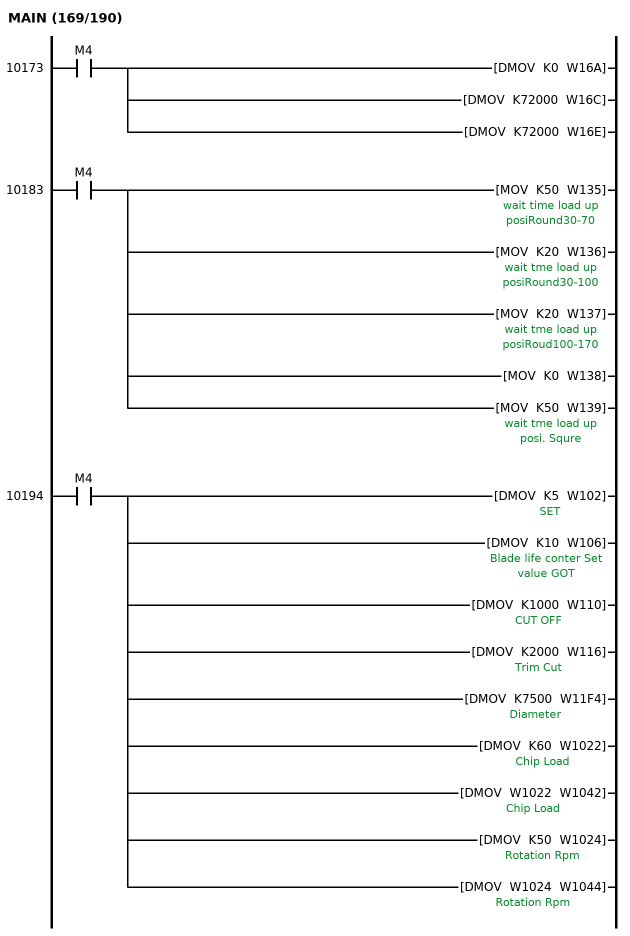
[picture p168: ladder of MAIN, rungs at steps 10173 to 10194]
10173 LD      M4
      DMOV    K0 W16A
      DMOV    K72000 W16C
      DMOV    K72000 W16E
10183 LD      M4
      MOV     K50 W135
      MOV     K20 W136
      MOV     K20 W137
      MOV     K0 W138
      MOV     K50 W139
10194 LD      M4
      DMOV    K5 W102
      DMOV    K10 W106
      DMOV    K1000 W110
      DMOV    K2000 W116
      DMOV    K7500 W11F4
      DMOV    K60 W1022
      DMOV    W1022 W1042
      DMOV    K50 W1024
      DMOV    W1024 W1044
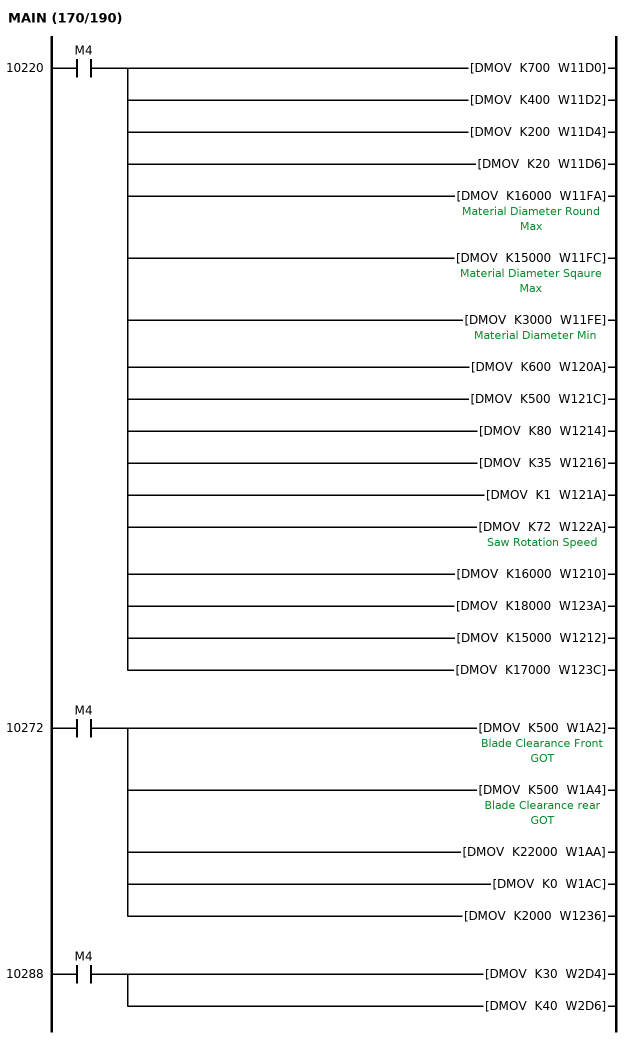
10220 LD      M4
      DMOV    K700 W11D0
      DMOV    K400 W11D2
      DMOV    K200 W11D4
      DMOV    K20 W11D6
      DMOV    K16000 W11FA
      DMOV    K15000 W11FC
      DMOV    K3000 W11FE
      DMOV    K600 W120A
      DMOV    K500 W121C
      DMOV    K80 W1214
      DMOV    K35 W1216
      DMOV    K1 W121A
      DMOV    K72 W122A
      DMOV    K16000 W1210
      DMOV    K18000 W123A
      DMOV    K15000 W1212
      DMOV    K17000 W123C
10272 LD      M4
      DMOV    K500 W1A2
      DMOV    K500 W1A4
      DMOV    K22000 W1AA
      DMOV    K0 W1AC
      DMOV    K2000 W1236
10288 LD      M4
      DMOV    K30 W2D4
      DMOV    K40 W2D6
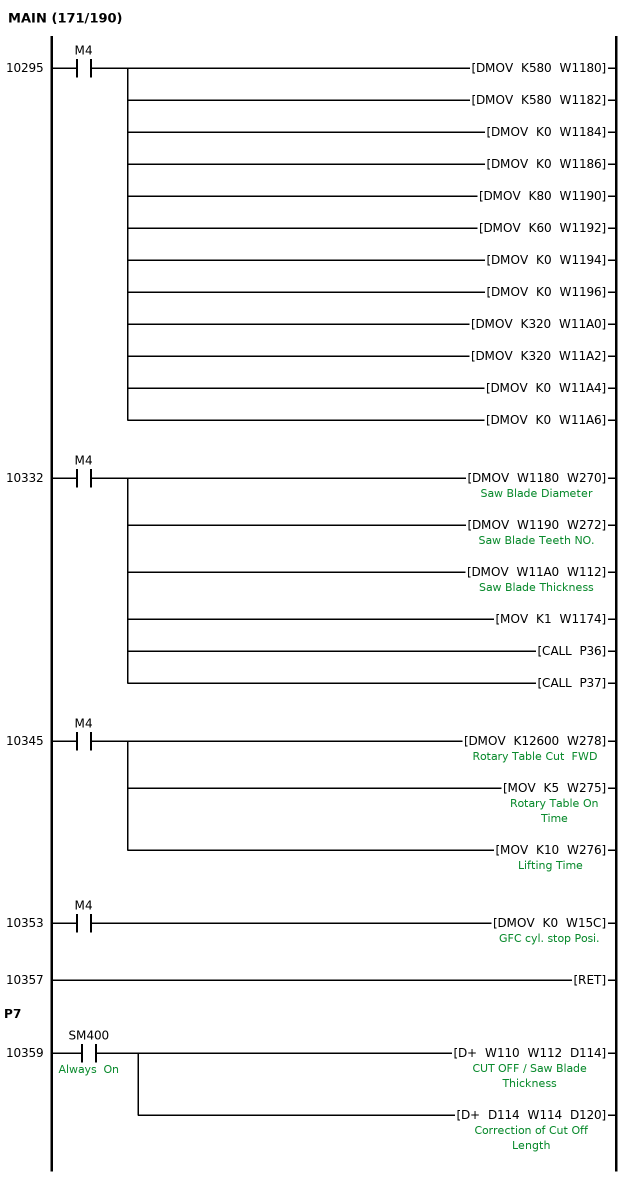
10295 LD      M4
      DMOV    K580 W1180
      DMOV    K580 W1182
      DMOV    K0 W1184
      DMOV    K0 W1186
      DMOV    K80 W1190
      DMOV    K60 W1192
      DMOV    K0 W1194
      DMOV    K0 W1196
      DMOV    K320 W11A0
      DMOV    K320 W11A2
      DMOV    K0 W11A4
      DMOV    K0 W11A6
10332 LD      M4
      DMOV    W1180 W270
      DMOV    W1190 W272
      DMOV    W11A0 W112
      MOV     K1 W1174
      CALL    P36
      CALL    P37
10345 LD      M4
      DMOV    K12600 W278
      MOV     K5 W275
      MOV     K10 W276
10353 LD      M4
      DMOV    K0 W15C  ; GFC cyl. stop Posi.
10357 RET
      P7
10359 LD      SM400  ; Always  On
      D+      W110 W112 D114
      D+      D114 W114 D120
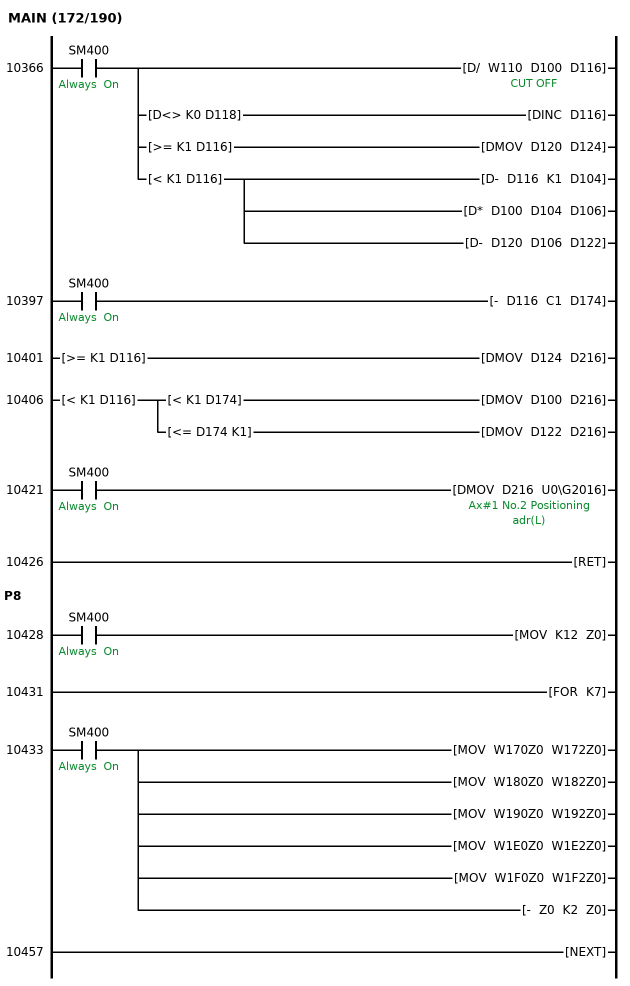
10366 LD      SM400  ; Always  On
      D/      W110 D100 D116
      MPS
      ANDD<>  K0 D118
      DINC    D116
      MRD
      AND>=   K1 D116
      DMOV    D120 D124
      MPP
      AND<    K1 D116
      D-      D116 K1 D104
      D*      D100 D104 D106
      D-      D120 D106 D122
10397 LD      SM400  ; Always  On
      -       D116 C1 D174
10401 LD>=    K1 D116
      DMOV    D124 D216
10406 LD<     K1 D116
      MPS
      AND<    K1 D174
      DMOV    D100 D216
      MPP
      AND<=   D174 K1
      DMOV    D122 D216
10421 LD      SM400  ; Always  On
      DMOV    D216 U0\G2016  ; Ax#1 No.2 Positioning adr(L)
10426 RET
      P8
10428 LD      SM400  ; Always  On
      MOV     K12 Z0
10431 FOR     K7
10433 LD      SM400  ; Always  On
      MOV     W170Z0 W172Z0
      MOV     W180Z0 W182Z0
      MOV     W190Z0 W192Z0
      MOV     W1E0Z0 W1E2Z0
      MOV     W1F0Z0 W1F2Z0
      -       Z0 K2 Z0
10457 NEXT
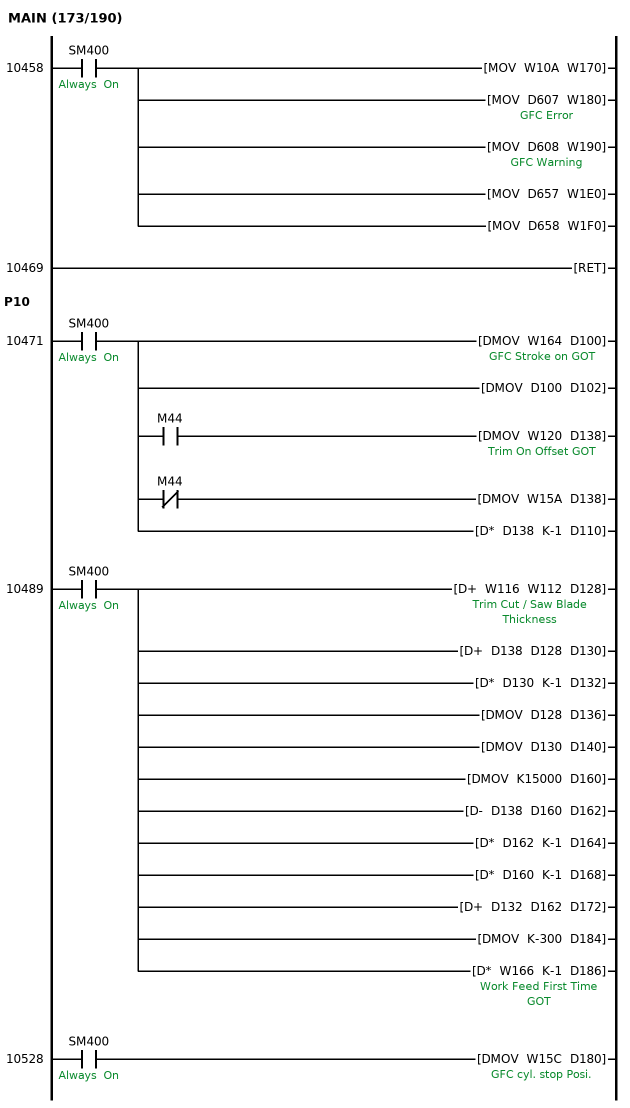
10458 LD      SM400  ; Always  On
      MOV     W10A W170
      MOV     D607 W180
      MOV     D608 W190
      MOV     D657 W1E0
      MOV     D658 W1F0
10469 RET
      P10
10471 LD      SM400  ; Always  On
      DMOV    W164 D100
      DMOV    D100 D102
      MPS
      AND     M44
      DMOV    W120 D138
      MRD
      ANI     M44
      DMOV    W15A D138
      MPP
      D*      D138 K-1 D110
10489 LD      SM400  ; Always  On
      D+      W116 W112 D128
      D+      D138 D128 D130
      D*      D130 K-1 D132
      DMOV    D128 D136
      DMOV    D130 D140
      DMOV    K15000 D160
      D-      D138 D160 D162
      D*      D162 K-1 D164
      D*      D160 K-1 D168
      D+      D132 D162 D172
      DMOV    K-300 D184
      D*      W166 K-1 D186
10528 LD      SM400  ; Always  On
      DMOV    W15C D180
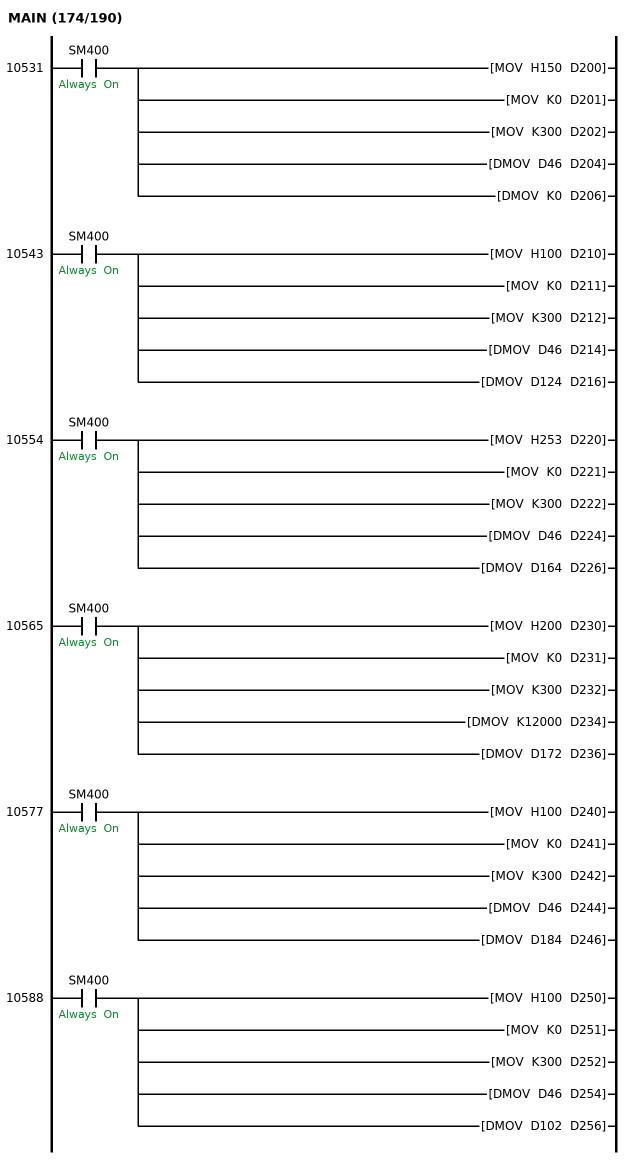
10531 LD      SM400  ; Always  On
      MOV     H150 D200
      MOV     K0 D201
      MOV     K300 D202
      DMOV    D46 D204
      DMOV    K0 D206
10543 LD      SM400  ; Always  On
      MOV     H100 D210
      MOV     K0 D211
      MOV     K300 D212
      DMOV    D46 D214
      DMOV    D124 D216
10554 LD      SM400  ; Always  On
      MOV     H253 D220
      MOV     K0 D221
      MOV     K300 D222
      DMOV    D46 D224
      DMOV    D164 D226
10565 LD      SM400  ; Always  On
      MOV     H200 D230
      MOV     K0 D231
      MOV     K300 D232
      DMOV    K12000 D234
      DMOV    D172 D236
10577 LD      SM400  ; Always  On
      MOV     H100 D240
      MOV     K0 D241
      MOV     K300 D242
      DMOV    D46 D244
      DMOV    D184 D246
10588 LD      SM400  ; Always  On
      MOV     H100 D250
      MOV     K0 D251
      MOV     K300 D252
      DMOV    D46 D254
      DMOV    D102 D256
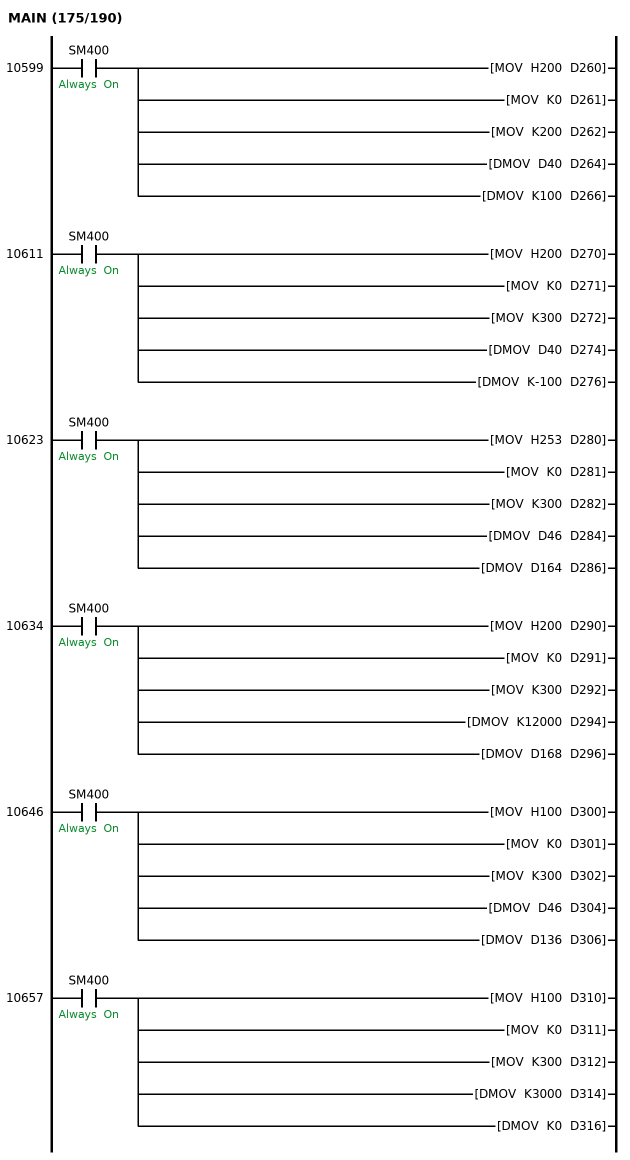
10599 LD      SM400  ; Always  On
      MOV     H200 D260
      MOV     K0 D261
      MOV     K200 D262
      DMOV    D40 D264
      DMOV    K100 D266
10611 LD      SM400  ; Always  On
      MOV     H200 D270
      MOV     K0 D271
      MOV     K300 D272
      DMOV    D40 D274
      DMOV    K-100 D276
10623 LD      SM400  ; Always  On
      MOV     H253 D280
      MOV     K0 D281
      MOV     K300 D282
      DMOV    D46 D284
      DMOV    D164 D286
10634 LD      SM400  ; Always  On
      MOV     H200 D290
      MOV     K0 D291
      MOV     K300 D292
      DMOV    K12000 D294
      DMOV    D168 D296
10646 LD      SM400  ; Always  On
      MOV     H100 D300
      MOV     K0 D301
      MOV     K300 D302
      DMOV    D46 D304
      DMOV    D136 D306
10657 LD      SM400  ; Always  On
      MOV     H100 D310
      MOV     K0 D311
      MOV     K300 D312
      DMOV    K3000 D314
      DMOV    K0 D316
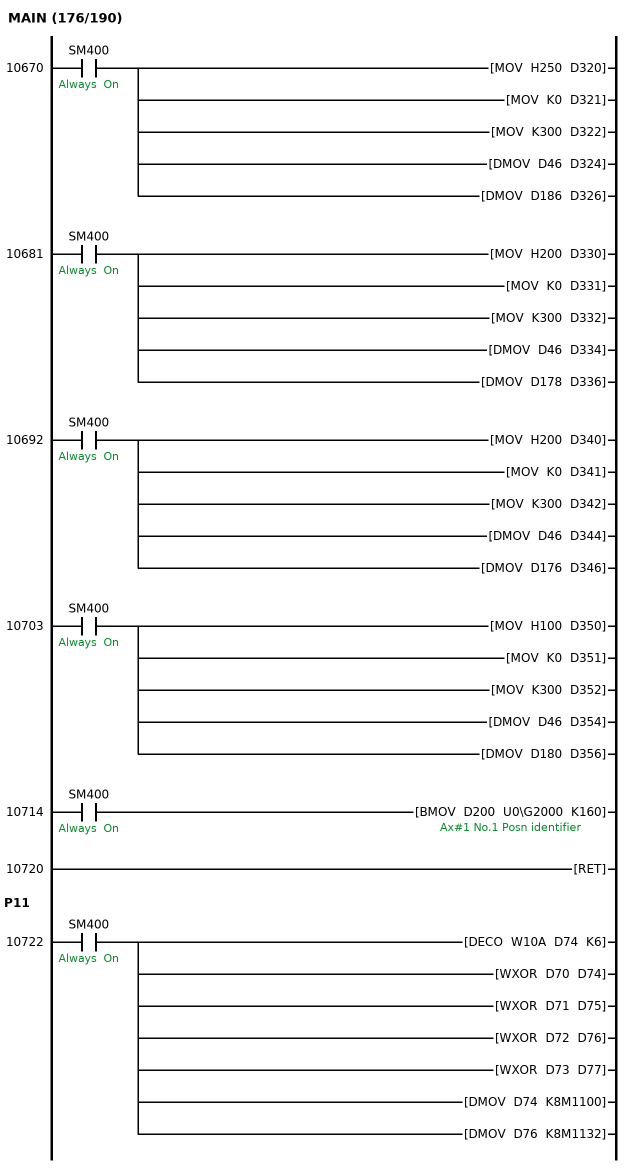
10670 LD      SM400  ; Always  On
      MOV     H250 D320
      MOV     K0 D321
      MOV     K300 D322
      DMOV    D46 D324
      DMOV    D186 D326
10681 LD      SM400  ; Always  On
      MOV     H200 D330
      MOV     K0 D331
      MOV     K300 D332
      DMOV    D46 D334
      DMOV    D178 D336
10692 LD      SM400  ; Always  On
      MOV     H200 D340
      MOV     K0 D341
      MOV     K300 D342
      DMOV    D46 D344
      DMOV    D176 D346
10703 LD      SM400  ; Always  On
      MOV     H100 D350
      MOV     K0 D351
      MOV     K300 D352
      DMOV    D46 D354
      DMOV    D180 D356
10714 LD      SM400  ; Always  On
      BMOV    D200 U0\G2000 K160  ; Ax#1 No.1 Posn identifier
10720 RET
      P11
10722 LD      SM400  ; Always  On
      DECO    W10A D74 K6
      WXOR    D70 D74
      WXOR    D71 D75
      WXOR    D72 D76
      WXOR    D73 D77
      DMOV    D74 K8M1100
      DMOV    D76 K8M1132
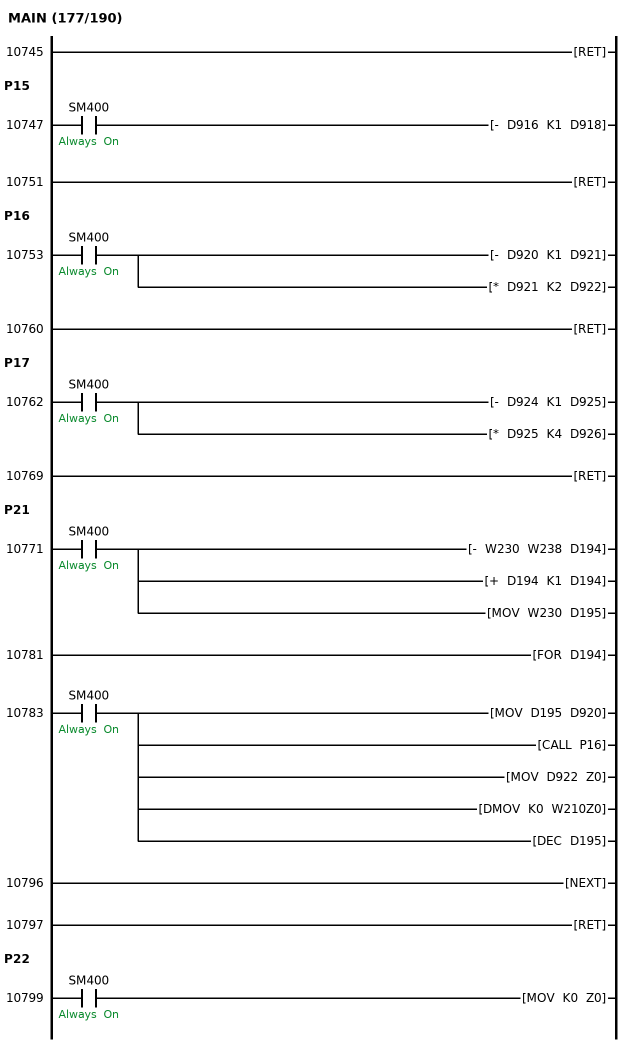
10745 RET
      P15
10747 LD      SM400  ; Always  On
      -       D916 K1 D918
10751 RET
      P16
10753 LD      SM400  ; Always  On
      -       D920 K1 D921
      *       D921 K2 D922
10760 RET
      P17
10762 LD      SM400  ; Always  On
      -       D924 K1 D925
      *       D925 K4 D926
10769 RET
      P21
10771 LD      SM400  ; Always  On
      -       W230 W238 D194
      +       D194 K1 D194
      MOV     W230 D195
10781 FOR     D194
10783 LD      SM400  ; Always  On
      MOV     D195 D920
      CALL    P16
      MOV     D922 Z0
      DMOV    K0 W210Z0
      DEC     D195
10796 NEXT
10797 RET
      P22
10799 LD      SM400  ; Always  On
      MOV     K0 Z0
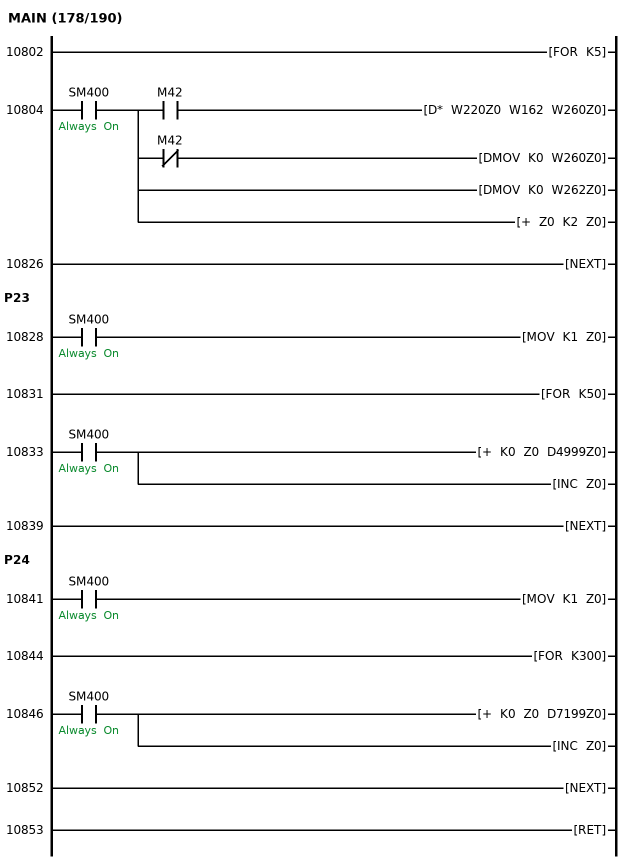
10802 FOR     K5
10804 LD      SM400  ; Always  On
      MPS
      AND     M42
      D*      W220Z0 W162 W260Z0
      MRD
      ANI     M42
      DMOV    K0 W260Z0
      MPP
      DMOV    K0 W262Z0
      +       Z0 K2 Z0
10826 NEXT
      P23
10828 LD      SM400  ; Always  On
      MOV     K1 Z0
10831 FOR     K50
10833 LD      SM400  ; Always  On
      +       K0 Z0 D4999Z0
      INC     Z0
10839 NEXT
      P24
10841 LD      SM400  ; Always  On
      MOV     K1 Z0
10844 FOR     K300
10846 LD      SM400  ; Always  On
      +       K0 Z0 D7199Z0
      INC     Z0
10852 NEXT
10853 RET
      P25
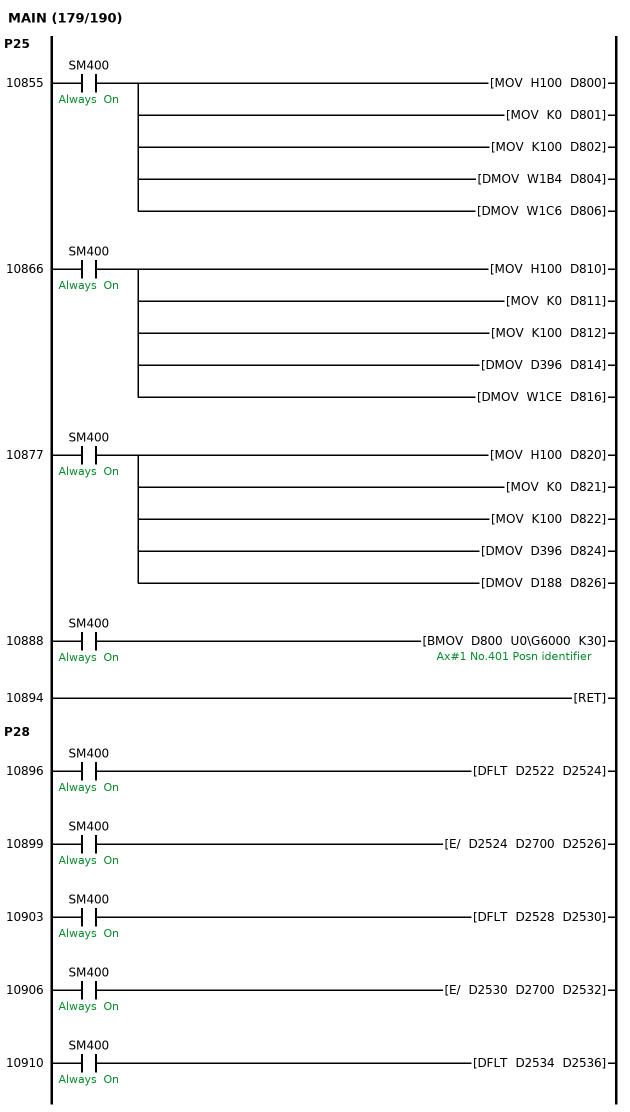
10855 LD      SM400  ; Always  On
      MOV     H100 D800
      MOV     K0 D801
      MOV     K100 D802
      DMOV    W1B4 D804
      DMOV    W1C6 D806
10866 LD      SM400  ; Always  On
      MOV     H100 D810
      MOV     K0 D811
      MOV     K100 D812
      DMOV    D396 D814
      DMOV    W1CE D816
10877 LD      SM400  ; Always  On
      MOV     H100 D820
      MOV     K0 D821
      MOV     K100 D822
      DMOV    D396 D824
      DMOV    D188 D826
10888 LD      SM400  ; Always  On
      BMOV    D800 U0\G6000 K30  ; Ax#1 No.401 Posn identifier
10894 RET
      P28
10896 LD      SM400  ; Always  On
      DFLT    D2522 D2524
10899 LD      SM400  ; Always  On
      E/      D2524 D2700 D2526
10903 LD      SM400  ; Always  On
      DFLT    D2528 D2530
10906 LD      SM400  ; Always  On
      E/      D2530 D2700 D2532
10910 LD      SM400  ; Always  On
      DFLT    D2534 D2536
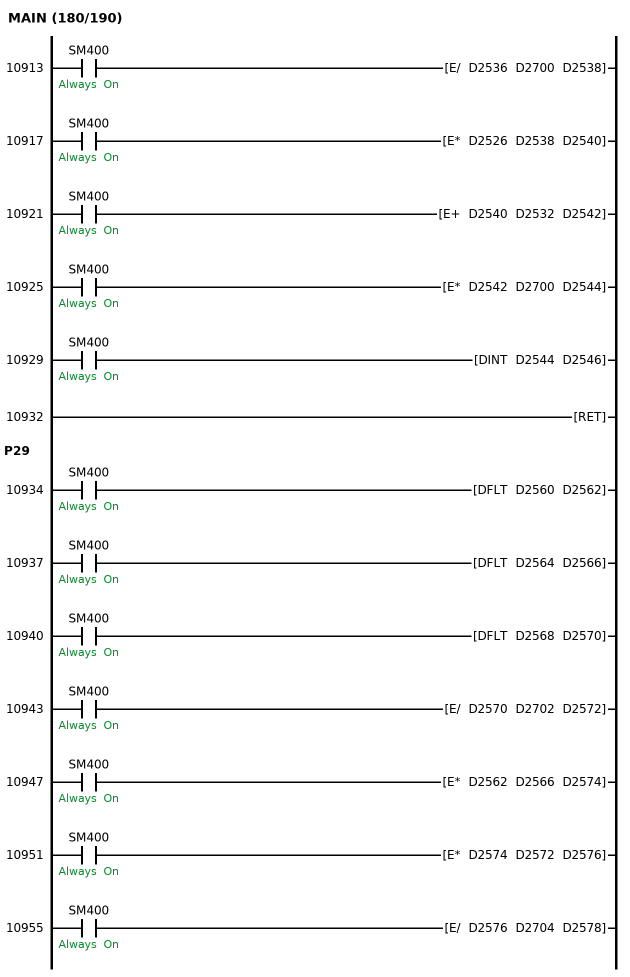
10913 LD      SM400  ; Always  On
      E/      D2536 D2700 D2538
10917 LD      SM400  ; Always  On
      E*      D2526 D2538 D2540
10921 LD      SM400  ; Always  On
      E+      D2540 D2532 D2542
10925 LD      SM400  ; Always  On
      E*      D2542 D2700 D2544
10929 LD      SM400  ; Always  On
      DINT    D2544 D2546
10932 RET
      P29
10934 LD      SM400  ; Always  On
      DFLT    D2560 D2562
10937 LD      SM400  ; Always  On
      DFLT    D2564 D2566
10940 LD      SM400  ; Always  On
      DFLT    D2568 D2570
10943 LD      SM400  ; Always  On
      E/      D2570 D2702 D2572
10947 LD      SM400  ; Always  On
      E*      D2562 D2566 D2574
10951 LD      SM400  ; Always  On
      E*      D2574 D2572 D2576
10955 LD      SM400  ; Always  On
      E/      D2576 D2704 D2578
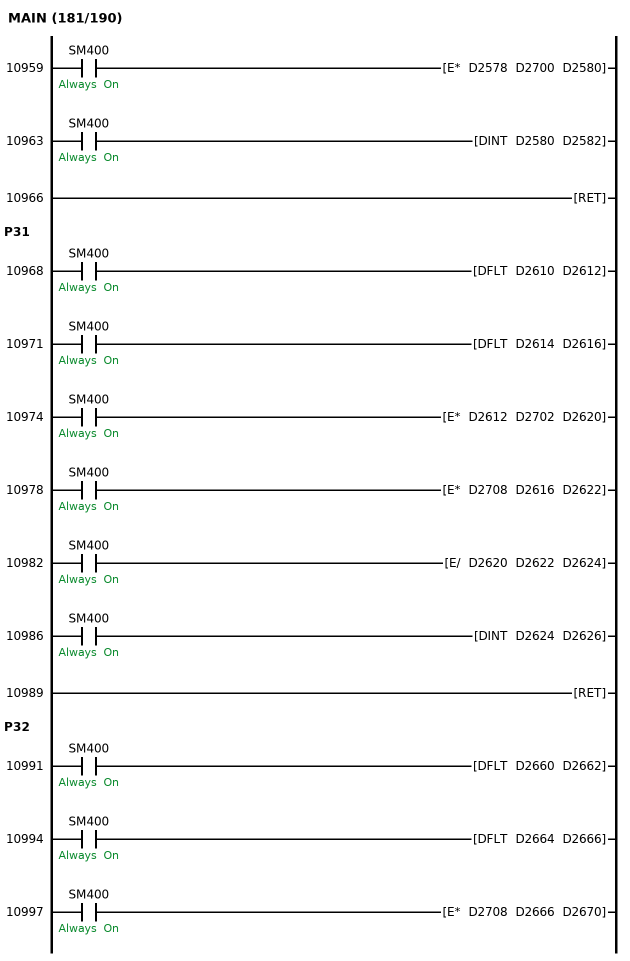
10959 LD      SM400  ; Always  On
      E*      D2578 D2700 D2580
10963 LD      SM400  ; Always  On
      DINT    D2580 D2582
10966 RET
      P31
10968 LD      SM400  ; Always  On
      DFLT    D2610 D2612
10971 LD      SM400  ; Always  On
      DFLT    D2614 D2616
10974 LD      SM400  ; Always  On
      E*      D2612 D2702 D2620
10978 LD      SM400  ; Always  On
      E*      D2708 D2616 D2622
10982 LD      SM400  ; Always  On
      E/      D2620 D2622 D2624
10986 LD      SM400  ; Always  On
      DINT    D2624 D2626
10989 RET
      P32
10991 LD      SM400  ; Always  On
      DFLT    D2660 D2662
10994 LD      SM400  ; Always  On
      DFLT    D2664 D2666
10997 LD      SM400  ; Always  On
      E*      D2708 D2666 D2670
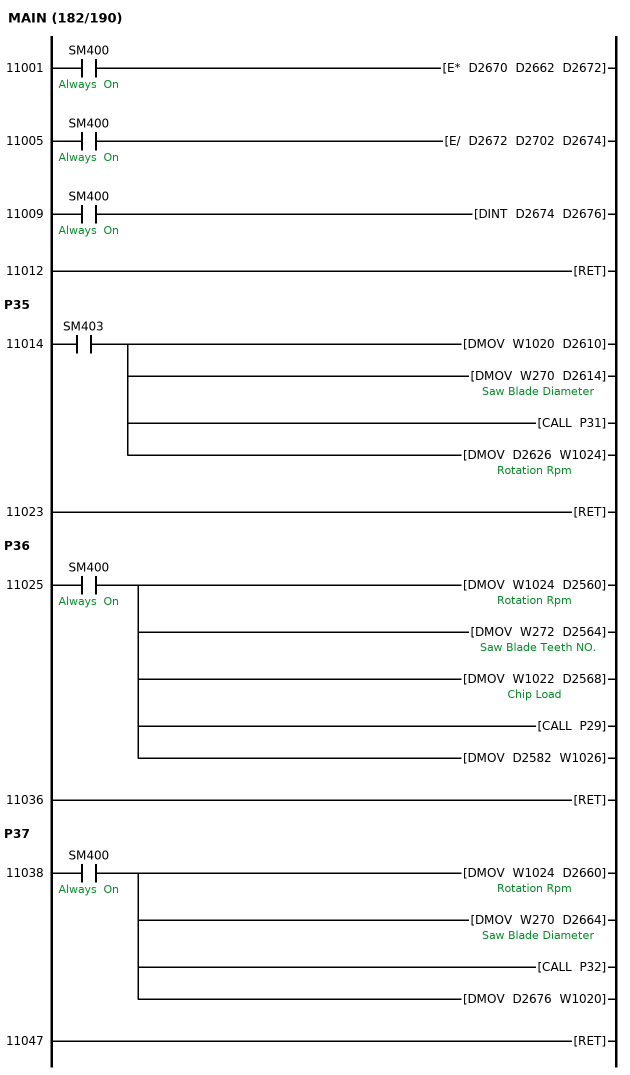
11001 LD      SM400  ; Always  On
      E*      D2670 D2662 D2672
11005 LD      SM400  ; Always  On
      E/      D2672 D2702 D2674
11009 LD      SM400  ; Always  On
      DINT    D2674 D2676
11012 RET
      P35
11014 LD      SM403
      DMOV    W1020 D2610
      DMOV    W270 D2614
      CALL    P31
      DMOV    D2626 W1024
11023 RET
      P36
11025 LD      SM400  ; Always  On
      DMOV    W1024 D2560
      DMOV    W272 D2564
      DMOV    W1022 D2568
      CALL    P29
      DMOV    D2582 W1026
11036 RET
      P37
11038 LD      SM400  ; Always  On
      DMOV    W1024 D2660
      DMOV    W270 D2664
      CALL    P32
      DMOV    D2676 W1020
11047 RET
      P40
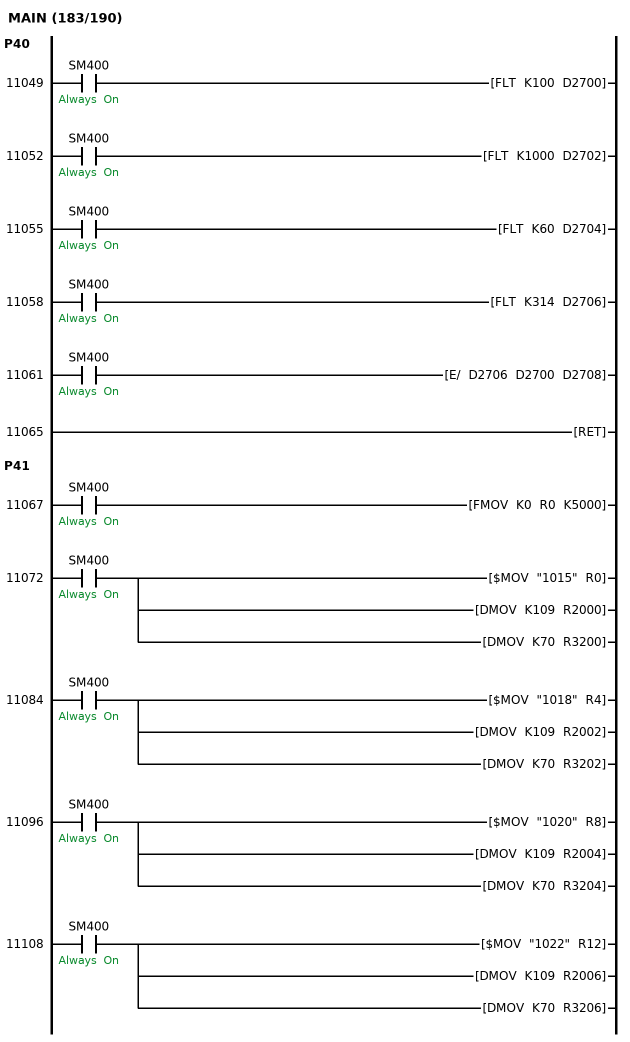
11049 LD      SM400  ; Always  On
      FLT     K100 D2700
11052 LD      SM400  ; Always  On
      FLT     K1000 D2702
11055 LD      SM400  ; Always  On
      FLT     K60 D2704
11058 LD      SM400  ; Always  On
      FLT     K314 D2706
11061 LD      SM400  ; Always  On
      E/      D2706 D2700 D2708
11065 RET
      P41
11067 LD      SM400  ; Always  On
      FMOV    K0 R0 K5000
11072 LD      SM400  ; Always  On
      $MOV    "1015" R0
      DMOV    K109 R2000
      DMOV    K70 R3200
11084 LD      SM400  ; Always  On
      $MOV    "1018" R4
      DMOV    K109 R2002
      DMOV    K70 R3202
11096 LD      SM400  ; Always  On
      $MOV    "1020" R8
      DMOV    K109 R2004
      DMOV    K70 R3204
11108 LD      SM400  ; Always  On
      $MOV    "1022" R12
      DMOV    K109 R2006
      DMOV    K70 R3206
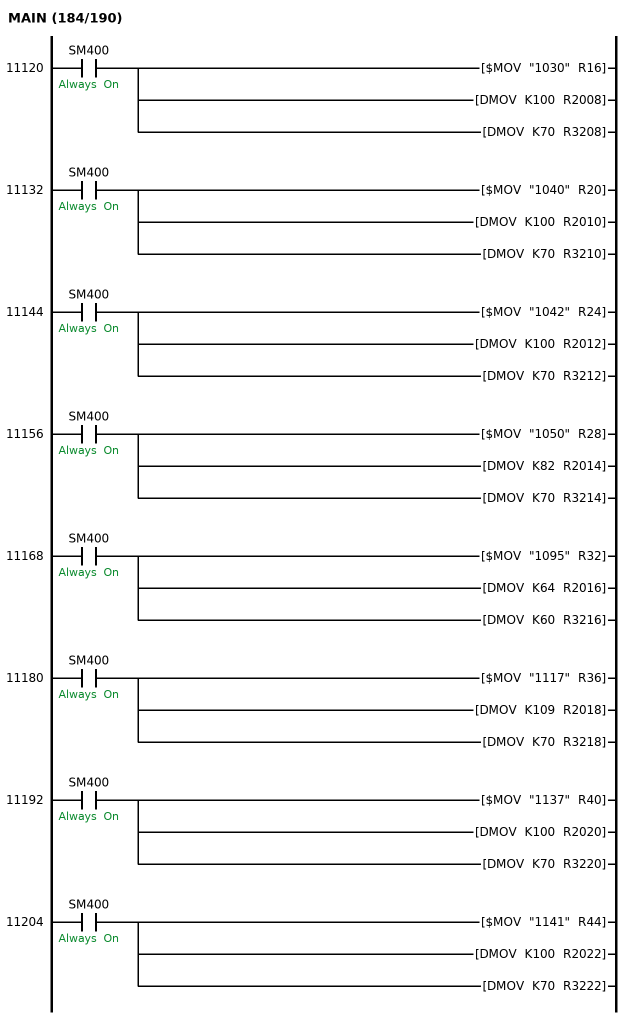
11120 LD      SM400  ; Always  On
      $MOV    "1030" R16
      DMOV    K100 R2008
      DMOV    K70 R3208
11132 LD      SM400  ; Always  On
      $MOV    "1040" R20
      DMOV    K100 R2010
      DMOV    K70 R3210
11144 LD      SM400  ; Always  On
      $MOV    "1042" R24
      DMOV    K100 R2012
      DMOV    K70 R3212
11156 LD      SM400  ; Always  On
      $MOV    "1050" R28
      DMOV    K82 R2014
      DMOV    K70 R3214
11168 LD      SM400  ; Always  On
      $MOV    "1095" R32
      DMOV    K64 R2016
      DMOV    K60 R3216
11180 LD      SM400  ; Always  On
      $MOV    "1117" R36
      DMOV    K109 R2018
      DMOV    K70 R3218
11192 LD      SM400  ; Always  On
      $MOV    "1137" R40
      DMOV    K100 R2020
      DMOV    K70 R3220
11204 LD      SM400  ; Always  On
      $MOV    "1141" R44
      DMOV    K100 R2022
      DMOV    K70 R3222
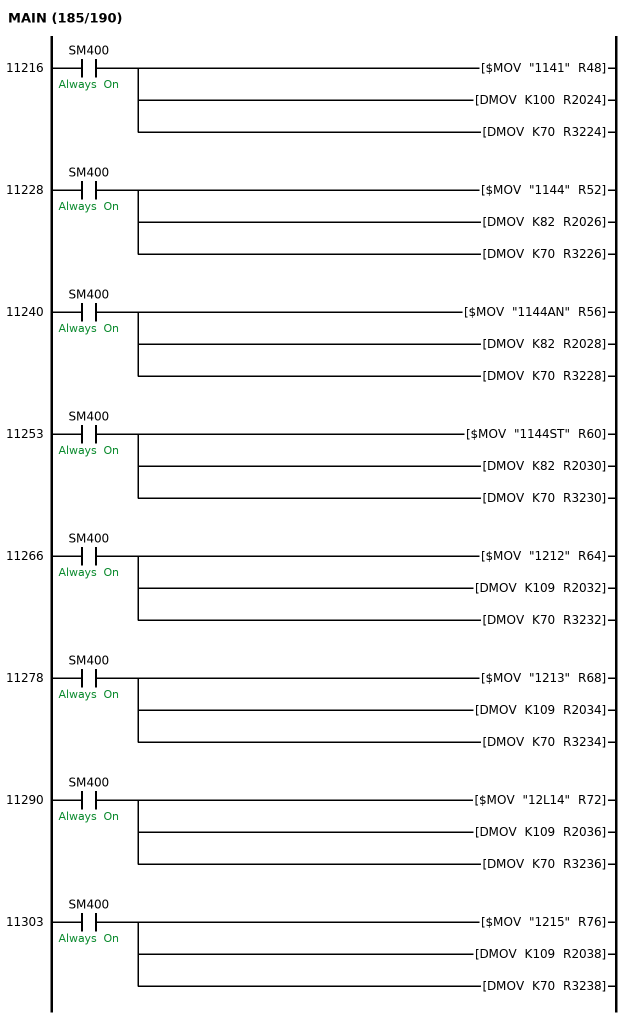
11216 LD      SM400  ; Always  On
      $MOV    "1141" R48
      DMOV    K100 R2024
      DMOV    K70 R3224
11228 LD      SM400  ; Always  On
      $MOV    "1144" R52
      DMOV    K82 R2026
      DMOV    K70 R3226
11240 LD      SM400  ; Always  On
      $MOV    "1144AN" R56
      DMOV    K82 R2028
      DMOV    K70 R3228
11253 LD      SM400  ; Always  On
      $MOV    "1144ST" R60
      DMOV    K82 R2030
      DMOV    K70 R3230
11266 LD      SM400  ; Always  On
      $MOV    "1212" R64
      DMOV    K109 R2032
      DMOV    K70 R3232
11278 LD      SM400  ; Always  On
      $MOV    "1213" R68
      DMOV    K109 R2034
      DMOV    K70 R3234
11290 LD      SM400  ; Always  On
      $MOV    "12L14" R72
      DMOV    K109 R2036
      DMOV    K70 R3236
11303 LD      SM400  ; Always  On
      $MOV    "1215" R76
      DMOV    K109 R2038
      DMOV    K70 R3238
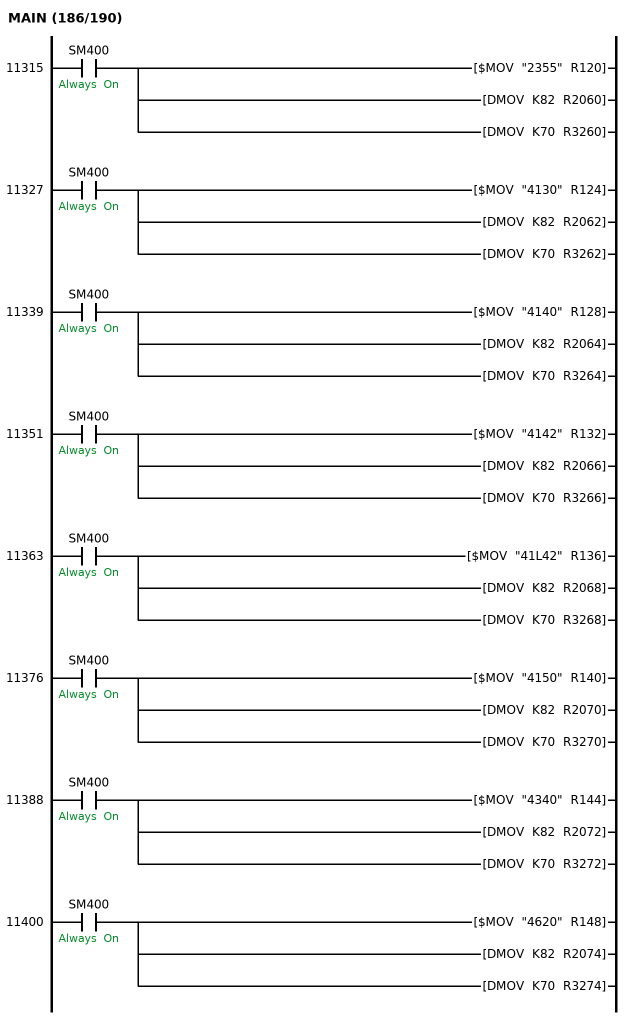
11315 LD      SM400  ; Always  On
      $MOV    "2355" R120
      DMOV    K82 R2060
      DMOV    K70 R3260
11327 LD      SM400  ; Always  On
      $MOV    "4130" R124
      DMOV    K82 R2062
      DMOV    K70 R3262
11339 LD      SM400  ; Always  On
      $MOV    "4140" R128
      DMOV    K82 R2064
      DMOV    K70 R3264
11351 LD      SM400  ; Always  On
      $MOV    "4142" R132
      DMOV    K82 R2066
      DMOV    K70 R3266
11363 LD      SM400  ; Always  On
      $MOV    "41L42" R136
      DMOV    K82 R2068
      DMOV    K70 R3268
11376 LD      SM400  ; Always  On
      $MOV    "4150" R140
      DMOV    K82 R2070
      DMOV    K70 R3270
11388 LD      SM400  ; Always  On
      $MOV    "4340" R144
      DMOV    K82 R2072
      DMOV    K70 R3272
11400 LD      SM400  ; Always  On
      $MOV    "4620" R148
      DMOV    K82 R2074
      DMOV    K70 R3274
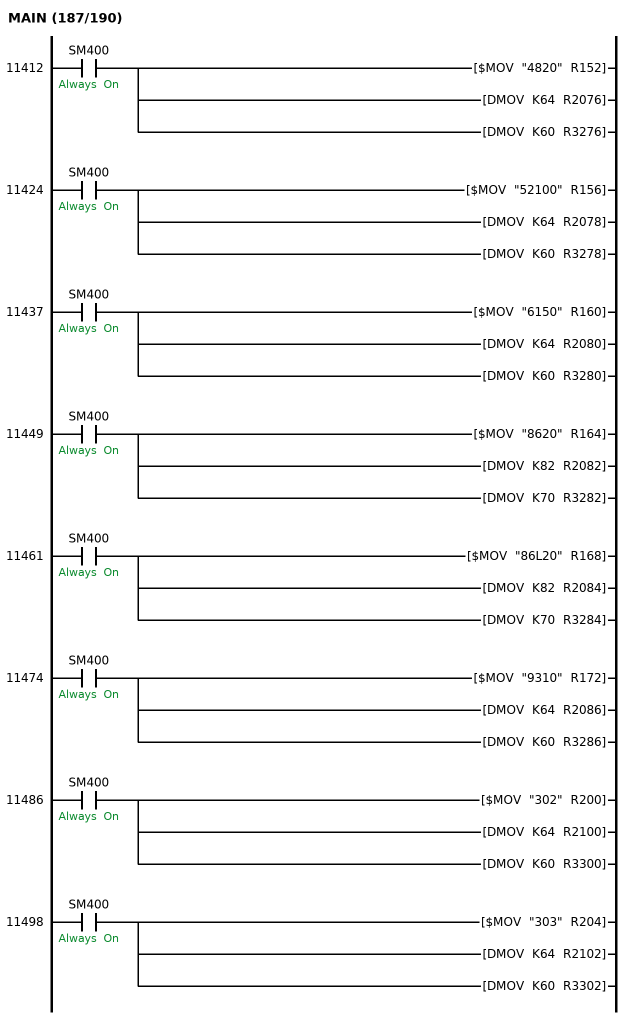
11412 LD      SM400  ; Always  On
      $MOV    "4820" R152
      DMOV    K64 R2076
      DMOV    K60 R3276
11424 LD      SM400  ; Always  On
      $MOV    "52100" R156
      DMOV    K64 R2078
      DMOV    K60 R3278
11437 LD      SM400  ; Always  On
      $MOV    "6150" R160
      DMOV    K64 R2080
      DMOV    K60 R3280
11449 LD      SM400  ; Always  On
      $MOV    "8620" R164
      DMOV    K82 R2082
      DMOV    K70 R3282
11461 LD      SM400  ; Always  On
      $MOV    "86L20" R168
      DMOV    K82 R2084
      DMOV    K70 R3284
11474 LD      SM400  ; Always  On
      $MOV    "9310" R172
      DMOV    K64 R2086
      DMOV    K60 R3286
11486 LD      SM400  ; Always  On
      $MOV    "302" R200
      DMOV    K64 R2100
      DMOV    K60 R3300
11498 LD      SM400  ; Always  On
      $MOV    "303" R204
      DMOV    K64 R2102
      DMOV    K60 R3302
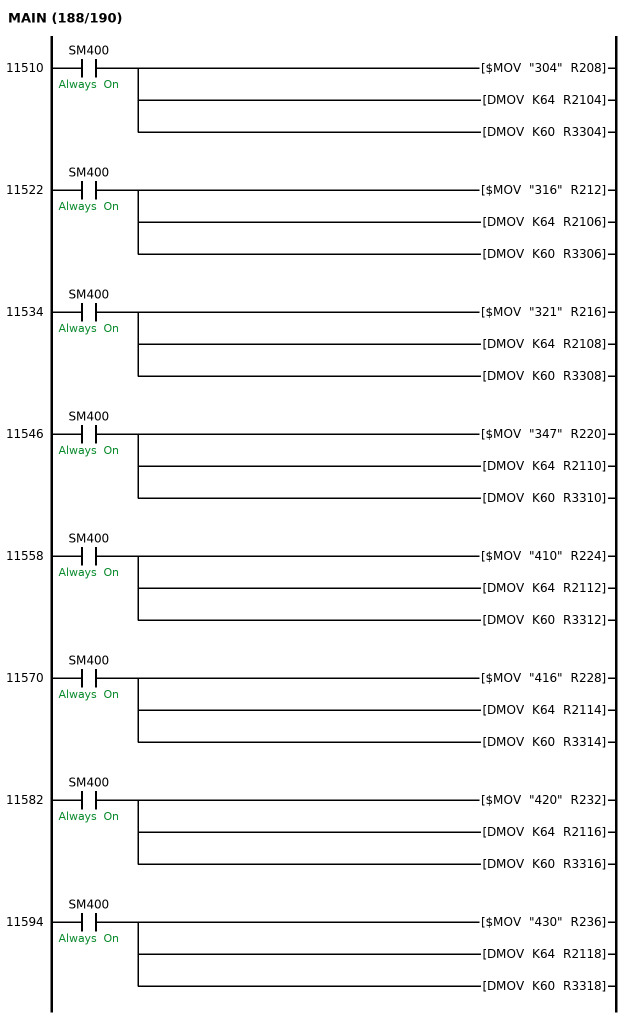
11510 LD      SM400  ; Always  On
      $MOV    "304" R208
      DMOV    K64 R2104
      DMOV    K60 R3304
11522 LD      SM400  ; Always  On
      $MOV    "316" R212
      DMOV    K64 R2106
      DMOV    K60 R3306
11534 LD      SM400  ; Always  On
      $MOV    "321" R216
      DMOV    K64 R2108
      DMOV    K60 R3308
11546 LD      SM400  ; Always  On
      $MOV    "347" R220
      DMOV    K64 R2110
      DMOV    K60 R3310
11558 LD      SM400  ; Always  On
      $MOV    "410" R224
      DMOV    K64 R2112
      DMOV    K60 R3312
11570 LD      SM400  ; Always  On
      $MOV    "416" R228
      DMOV    K64 R2114
      DMOV    K60 R3314
11582 LD      SM400  ; Always  On
      $MOV    "420" R232
      DMOV    K64 R2116
      DMOV    K60 R3316
11594 LD      SM400  ; Always  On
      $MOV    "430" R236
      DMOV    K64 R2118
      DMOV    K60 R3318
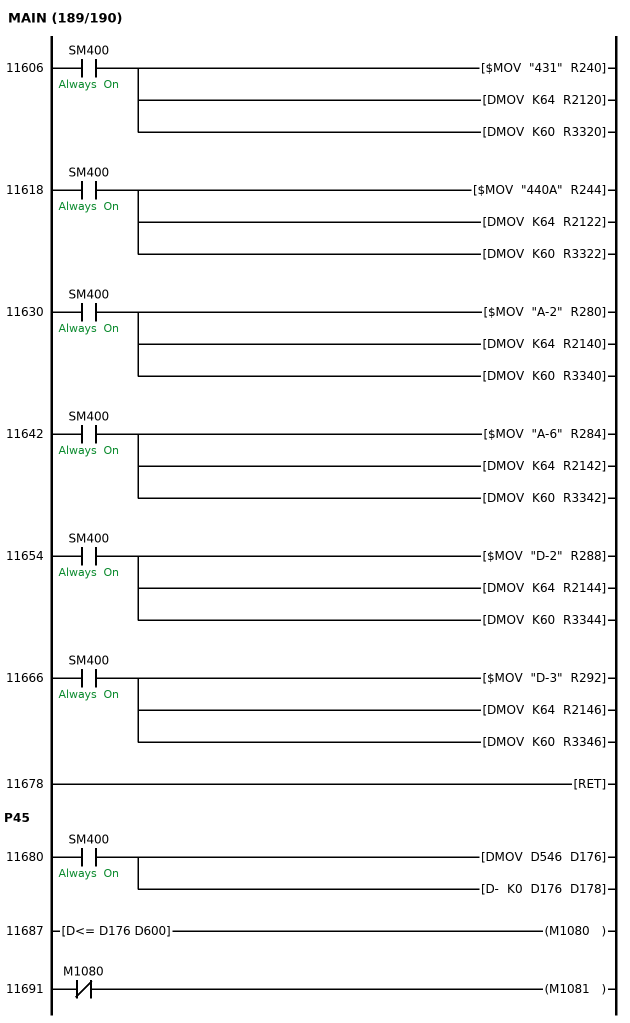
11606 LD      SM400  ; Always  On
      $MOV    "431" R240
      DMOV    K64 R2120
      DMOV    K60 R3320
11618 LD      SM400  ; Always  On
      $MOV    "440A" R244
      DMOV    K64 R2122
      DMOV    K60 R3322
11630 LD      SM400  ; Always  On
      $MOV    "A-2" R280
      DMOV    K64 R2140
      DMOV    K60 R3340
11642 LD      SM400  ; Always  On
      $MOV    "A-6" R284
      DMOV    K64 R2142
      DMOV    K60 R3342
11654 LD      SM400  ; Always  On
      $MOV    "D-2" R288
      DMOV    K64 R2144
      DMOV    K60 R3344
11666 LD      SM400  ; Always  On
      $MOV    "D-3" R292
      DMOV    K64 R2146
      DMOV    K60 R3346
11678 RET
      P45
11680 LD      SM400  ; Always  On
      DMOV    D546 D176
      D-      K0 D176 D178
11687 LDD<=   D176 D600
      OUT     M1080
11691 LDI     M1080
      OUT     M1081
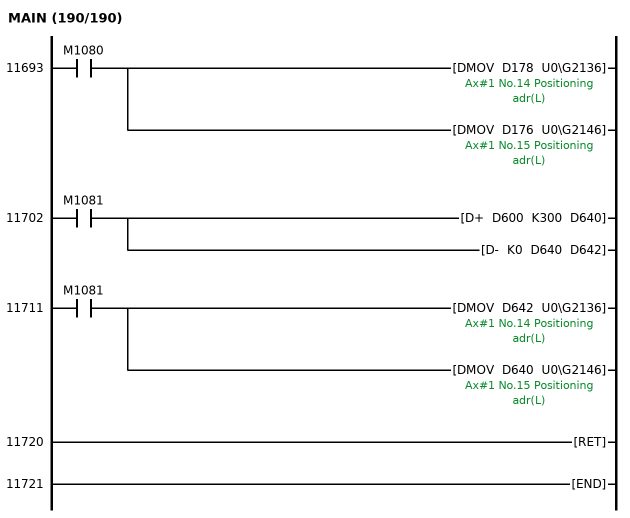
11693 LD      M1080
      DMOV    D178 U0\G2136  ; Ax#1 No.14 Positioning adr(L)
      DMOV    D176 U0\G2146  ; Ax#1 No.15 Positioning adr(L)
11702 LD      M1081
      D+      D600 K300 D640
      D-      K0 D640 D642
11711 LD      M1081
      DMOV    D642 U0\G2136
      DMOV    D640 U0\G2146
11720 RET
11721 END
END_PROGRAM

// device comments not shown above
X4  ; Ax#1 M code ON
X5  ; Ax#2 M code ON
X0A5  ; Material Stop
X0A8  ; Completion of material Throughin
X0AB  ; HYD ON IL PB
X0AC  ; HYD Auto Loader ON
X0BE  ; Rotary Table ON
X0BF  ; Local/ Remote
B201  ; Saw Head Fwd/Bwd  Enable
B202  ; GFC Wise Clamp/Unclamp Enable
B203  ; GFC feed Fwd/Bwd Enable
B204  ; Lader Up/Dn enable
B205  ; Work Stop Fwd/Bwd Enable
B206  ; Float wise On/Off Enable
B207  ; Float work On/Off Enable
B208  ; Seperation Trim/work Enable
B20B  ; Mist ON/Off Enable
B20C  ; Air Blow On/Off Enable
B210  ; Rotary Table fwd/ bwd  Enable
B211  ; Rotary Table ON/ OFF  Enable
B212  ; Lifting Enable
B10AB  ; Warning
Y14  ; Ax#1 Execution prohibition flag
Y15  ; Ax#2 Execution prohibition flag
Y9E  ; Auto Cycle ON
Y9F  ; Ready
